// TIA Portal V18 export
// export: Created 2026-01-09T11:23:25.5921821Z, ExportSetting WithDefaults, DisplayName Totally Integrated Automation Portal, DisplayVersion V18 Update 5, DisplayName TIA Portal Openness, DisplayVersion V18 Update 5, DisplayName TIA Portal Teamcenter Gateway, DisplayVersion V18, DisplayName TIA Portal Version Control Interface, DisplayVersion V18, DisplayName SINAMICS Startdrive Advanced, DisplayVersion V18 SP2 Update 1, DisplayName SINAMICS Startdrive G110M, G120, G120C, G120D, G120P, G115D, DisplayVersion V18 SP2 Update 1, DisplayName SINAMICS Startdrive G130, G150, S120, S150, SINAMICS MV, S210, G220, S200, DisplayVersion V18 SP2 Update 1, DisplayName STEP 7 Professional, DisplayVersion V18 Update 5, DisplayName STEP 7 Safety, DisplayVersion V18, DisplayName WinCC Professional, DisplayVersion V18 Update 5
Screen "123ProcessValue2"  1280x800, Number=123, Template=01Auto
  ScreenLayer 
    FaceplateInstance "Process_Data_1" at 10,89 size 425x285  FaceplateTypeName=ProcessData@$@Process_Data V 0.0.14
      Property_1 := AutoProcessData_F_Robot2Grip2
      InterfacePropertyText "Name_t"  Text="F_Robot2Grip2"
    FaceplateInstance "Process_Data_2" at 430,89 size 425x285  FaceplateTypeName=ProcessData@$@Process_Data V 0.0.14
      Property_1 := AutoProcessData_C_GlueNGBuffer
      InterfacePropertyText "Name_t"  Text="GlueNGBuffer"
    FaceplateInstance "Process_Data_3" at 850,89 size 425x285  FaceplateTypeName=ProcessData@$@Process_Data V 0.0.14
      Property_1 := AutoProcessData_C_MagnScanNGBuffer
      InterfacePropertyText "Name_t"  Text="MagnScanNGBuffer"
    FaceplateInstance "Process_Data_4" at 10,388 size 425x285  FaceplateTypeName=ProcessData@$@Process_Data V 0.0.14
      Property_1 := AutoProcessData_B_Press2
      InterfacePropertyText "Name_t"  Text="B_Press2"
    FaceplateInstance "Process_Data_5" at 430,388 size 425x285  FaceplateTypeName=ProcessData@$@Process_Data V 0.0.14
      Property_1 := AutoProcessData_F_Robot3Grip1
      InterfacePropertyText "Name_t"  Text="F_Robot3Grip1"
    FaceplateInstance "Process_Data_6" at 850,388 size 425x285  FaceplateTypeName=ProcessData@$@Process_Data V 0.0.14
      Property_1 := AutoProcessData_F_Robot3Grip2
      InterfacePropertyText "Name_t"  Text="F_Robot3Grip2"
    Button "btnMenu7_1" at 767,725 size 128x75  Mode=Text, StyleItem=BtnActive18, TextOff="过程 数据2 / Process Data_2 / Procesné data 2", TextOn="过程 数据2 / Process Data_2 / Procesné data 2"
      on Click: ActivateScreen(Screen name := , Object number := 0); SetTag(Tag := Sys_VersionManagement_HMIPageID, Value := 123)
    Button "btnMenu6" at 640,725 size 128x75  Mode=Text, StyleItem=BtnNormal20, TextOff="过程 数据1 / Process Data_1 / Procesné data 1", TextOn="过程 数据1 / Process Data_1 / Procesné data 1"
      on Click: ActivateScreen(Screen name := 123ProcessValue1, Object number := 0); SetTag(Tag := Sys_VersionManagement_HMIPageID, Value := 123)
    Button "btnMenu6_1" at 512,725 size 128x75  Mode=Text, StyleItem=BtnNormal20, TextOff="工装 扫码数据 / Tooling ScanData / Prípravok Scan Data", TextOn="工装 扫码数据 / Tooling ScanData / Nástroje Scan Data"
      on Click: ActivateScreen(Screen name := 125ProcessValue3, Object number := 0); SetTag(Tag := Sys_VersionManagement_HMIPageID, Value := 125)
    Button "btnMenu7_3" at 896,725 size 128x75  Mode=Text, StyleItem=BtnNormal20, TextOff="过程 数据Buffer / Process Data_Buffer", TextOn="过程 数据Buffer / Process Data_Buffer"
      on Click: ActivateScreen(Screen name := 129ProcessValue_Buffer, Object number := 0); SetTag(Tag := Sys_VersionManagement_HMIPageID, Value := 129)
